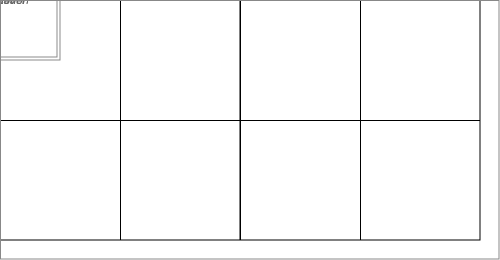
VISUALIZATION VisuLayout  // 500x260
    Group (0,0 240x240)
        Rectangle (0,0 240x240)
        Line (120,0) (120,240)
        Line (0,120) (240,120)
    Group (240,0 240x240)
        Rectangle (0,0 240x240)
        Line (120,0) (120,240)
        Line (0,120) (240,120)
    Frame (-60,-60 120x120)
        shows VisuStation(j := 1)
    Frame (-60,-60 120x120)
        shows VisuStation(j := 2)
    Frame (-60,-60 120x120)
        shows VisuStation(j := 3)
    Frame (-57,-57 114x114)
        shows VisuMover(i := 1)
    Frame (-57,-57 114x114)
        shows VisuMover(i := 2)
    Frame (-57,-57 114x114)
        shows VisuMover(i := 3)
END_VISUALIZATION

(* stored: Version 1.1.0.1, ProductVersion 3.1.4024.12
   Visu VisuLayout: Id {eac48a93-2837-44a2-85bc-1846388c48aa} *)
